FUNCTION f_ReservoirConvectionHeat : REAL
VAR_INPUT
	ReservoirTemperature : REAL ; // Celcius
	AmbientTemperature : REAL ; // Celcius
END_VAR
VAR_OUTPUT
	ReservoirConvectionHeat: REAL ; // Watt
END_VAR
VAR
	ConvectiveHeatTransferCoeff : REAL := 10 ; // Watt/(m2 K)
	ReservoirSurfaceArea : REAL :=6 ; // m2
END_VAR

f_ReservoirConvectionHeat := ConvectiveHeatTransferCoeff * ReservoirSurfaceArea * (ReservoirTemperature - AmbientTemperature);

END_FUNCTION

(* stored: Version 1.1.0.1, ProductVersion 3.1.4024.12
   POU f_ReservoirConvectionHeat: Id {d594b84b-0994-40e4-b68c-d2f887787c43}, SpecialFunc None *)
